Universal Robots URScript: test2.urscript

def test():

movej([0, -1.5708, -1.5708, -1.5708, 0, 0],a=0.1,v=0.05)

end
